FUNCTION_BLOCK FB_SoftWash IMPLEMENTS I_WashStrategy

VAR
	
	nRinseCount : INT := 1;
	iMotorRef : I_Motor;
	bWashing : BOOL;
	bDrying : BOOL;
	
	tWashTime : TIME := T#5S;
	nMotorWashSpeed : INT := 100;
	
	nMotorDrySpeed : INT := 700; 
	nMotorDryTime : TIME := T#7S;
	
	fbWashTimer : TON;
END_VAR

{warning 'add method implementation '}
METHOD GetDuration : TIME
VAR
END_VAR
GetDuration := tWashTime * (nRinseCount+1) + nMotorDryTime ;
END_METHOD

METHOD GetRinseCount : INT
VAR_INPUT
END_VAR
GetRinseCount := nRinseCount+1;
END_METHOD

METHOD StartSpin : BOOL
bDrying := TRUE;
fbWashTimer( IN := bDrying, PT := nMotorDryTime);
IF NOT fbWashTimer.Q THEN
	iMotorRef.DrySpin(nMotorDrySpeed);
ELSE
	iMotorRef.Stop();
	bDrying := FALSE;
	fbWashTimer( IN := bDrying);
	StartSpin := TRUE;
END_IF
END_METHOD

{warning 'add method implementation '}
METHOD StartWash : BOOL
VAR_INPUT
	iMotor : I_Motor;
END_VAR
iMotorRef := iMotor;
bWashing := TRUE;
fbWashTimer( IN := bWashing, PT := tWashTime);
IF NOT fbWashTimer.Q THEN
	iMotorRef.WashSpin(nMotorWashSpeed);
ELSE
	iMotorRef.Stop();
	bWashing := FALSE;
	fbWashTimer( IN := bWashing);
	StartWash := TRUE;
END_IF
END_METHOD

{warning 'add method implementation '}
METHOD Stop
bWashing := FALSE;
END_METHOD

END_FUNCTION_BLOCK

(* stored: Version 1.1.0.1, ProductVersion 3.1.4024.16
   POU FB_SoftWash: Id {db75bac4-9ece-4aa1-ad1b-7ea85c57614e}, SpecialFunc None
   Method GetDuration: Id {5610f62e-d353-4b19-81ab-f8bc1457e3bd}
   Method GetRinseCount: Id {a4f0e20d-04de-4f2a-9742-23b6eaab6815}
   Method StartSpin: Id {0bc1b6f3-2a77-45d0-8b68-67eb4e57f35a}
   Method StartWash: Id {1fc56eb1-f0aa-426e-a966-3c9d946c4f4e}
   Method Stop: Id {35f600ee-1d7f-4132-bc7c-9dbc289bcc2e} *)
